FUNCTION Runtime
VAR_STAT
	bInit	: BOOL := TRUE;
END_VAR

IF bInit THEN
	_Runtime.iFirstInit.Init();
	bInit := FALSE;
END_IF

IF _Runtime.iFirstCyclic <> 0 THEN
	_Runtime.iFirstCyclic.Exe();
END_IF

END_FUNCTION

(* stored: Version 1.1.0.1
   POU Runtime: Id {57f056fa-9062-499a-a7e4-db28982dc70c}, SpecialFunc None *)
